Universal Robots PolyScope program: external_control.urp

Program external_control2 (installation=default directory=/home/mahp/ursim-5.9.4.1031232/programs createdIn=5.9.4.1031232 lastSavedIn=5.9.4.1031232 robotSerialNumber=20195599999)
Calibrated DH parameters: a=[0, -0.425, -0.3922, 0, 0, 0]; d=[0.1625, 0, 0, 0.1333, 0.0997, 0.0996]; alpha=[1.570796, 0, 0, 1.570796, -1.570796, 0]; deltaTheta=[0, 0, 0, 0, 0, 0]
Robot Program (runOnlyOnce=false)
  URCap External Control (External Control, FZI Research Center for Information Technology)
